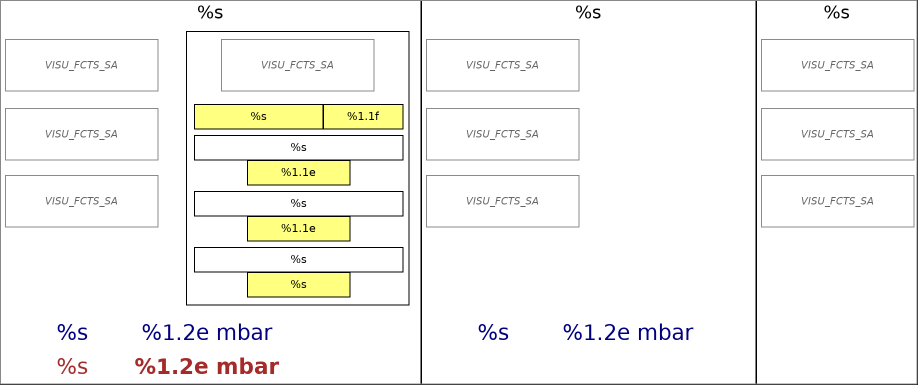
VISUALIZATION SA_POMP_2E_PCR_PPM_ASS  // 918x385
VAR_IN_OUT
	m_Input_PRG:			BLOCK_PRG_POMPAGE;
	m_Input_Jauge:			BLOCK_BCG450_ETHERCAT;
	m_Input_Process:		BLOCK_CDG_ETHERCAT;
	m_Input_Pr_Sas:			BLOCK_PCG550_ETHERCAT;
	m_Input_Vanne:			BLOCK_VVAT_650_ETHERCAT;
	m_Input_Machine:		BLOCK_MODE_MARCHE;
END_VAR
    Rectangle (0,0 421x385), "%s", text list: 'TextList_Navigation', text index: 6
    Rectangle (421,0 335x385), "%s", text list: 'TextList_Navigation', text index: 7
    Rectangle (756,0 162x385), "%s", text list: 'TextList_Navigation', text index: 13
    Frame (761,39 153x52)
        shows VISU_FCTS_SA(m_Input_ID_XML := 1, m_Input_UserRight := PRG_USER.ACTU_USER.FONCTION_SA, m_Input_Operation := m_Input_PRG.POMPAGE.OP_Marche_Pompes)
    Frame (761,108 153x52)
        shows VISU_FCTS_SA(m_Input_ID_XML := 2, m_Input_UserRight := PRG_USER.ACTU_USER.FONCTION_SA, m_Input_Operation := m_Input_PRG.POMPAGE.OP_Arret_Pompes)
    Rectangle (41,320 63x25), "%s", text variable: m_Input_Jauge.MNEMO
    Rectangle (111,318 192x29), "%1.2e mbar", text variable: m_Input_Jauge.STATE_Pression
    Rectangle (41,354 63x25), "%s", text variable: m_Input_Process.MNEMO
    Rectangle (111,352 192x29), "%1.2e mbar", text variable: m_Input_Process.STATE_Pression
    Frame (5,39 153x52)
        shows VISU_FCTS_SA(m_Input_ID_XML := 0, m_Input_UserRight := PRG_USER.ACTU_USER.FONCTION_SA, m_Input_Operation := m_Input_PRG.POMPAGE.OP_Pompage_Sec)
    Frame (426,39 153x52)
        shows VISU_FCTS_SA(m_Input_ID_XML := 0, m_Input_UserRight := PRG_USER.ACTU_USER.PRODUCTION, m_Input_Operation := m_Input_PRG.POMPAGE.OP_Pompage_SAS)
    Frame (5,108 153x52)
        shows VISU_FCTS_SA(m_Input_ID_XML := 3, m_Input_UserRight := PRG_USER.ACTU_USER.FONCTION_SA, m_Input_Operation := m_Input_PRG.POMPAGE.OP_Isolement)
    Frame (426,108 153x52)
        shows VISU_FCTS_SA(m_Input_ID_XML := 3, m_Input_UserRight := PRG_USER.ACTU_USER.FONCTION_SA, m_Input_Operation := m_Input_PRG.POMPAGE.OP_Isolement_SAS)
    Frame (761,175 153x52)
        shows VISU_FCTS_SA(m_Input_ID_XML := 17, m_Input_UserRight := PRG_USER.ACTU_USER.FONCTION_SA, m_Input_Operation := m_Input_PRG.POMPAGE.OP_Regen)
    Frame (5,175 153x52)
        shows VISU_FCTS_SA(m_Input_ID_XML := 4, m_Input_UserRight := PRG_USER.ACTU_USER.FONCTION_SA, m_Input_Operation := m_Input_PRG.POMPAGE.OP_Ventilation)
    Frame (426,175 153x52)
        shows VISU_FCTS_SA(m_Input_ID_XML := 4, m_Input_UserRight := PRG_USER.ACTU_USER.PRODUCTION, m_Input_Operation := m_Input_PRG.POMPAGE.OP_Ventilation_SAS)
    Rectangle (462,320 63x25), "%s", text variable: m_Input_Pr_Sas.MNEMO
    Rectangle (532,318 192x29), "%1.2e mbar", text variable: m_Input_Pr_Sas.STATE_Pression
    Rectangle (186,31 223x274)
    Frame (221,39 153x52)
        shows VISU_FCTS_SA(m_Input_ID_XML := 11, m_Input_UserRight := PRG_USER.ACTU_USER.FONCTION_SA, m_Input_Operation := m_Input_PRG.POMPAGE.OP_Pompage_Proc)
    RoundedRectangle (194,104 129x25), "%s", invisible if: NOT m_Input_Vanne.PRM_Mode, input disabled if: NOT (PRG_USER.ACTU_USER.FONCTION_SA AND NOT m_Input_MACHINE.STATE_Prod) OR m_Input_MACHINE.STATE_Prod, text list: 'TextList_VVAT_650_ETHERCAT', text index: 8
        OnMouseClick: toggle m_Input_Vanne.PRM_Mode
    RoundedRectangle (194,104 129x25), "%s", invisible if: m_Input_Vanne.PRM_Mode, input disabled if: NOT (PRG_USER.ACTU_USER.FONCTION_SA AND NOT m_Input_MACHINE.STATE_Prod) OR m_Input_MACHINE.STATE_Prod, text list: 'TextList_VVAT_650_ETHERCAT', text index: 7
        OnMouseClick: toggle m_Input_Vanne.PRM_Mode
    RoundedRectangle (194,135 209x25), "%s", invisible if: NOT m_Input_Vanne.PRM_Mode, text list: 'TextList_VVAT_650_ETHERCAT', text index: 4
    RoundedRectangle (194,191 209x25), "%s", invisible if: NOT m_Input_Vanne.PRM_Mode, text list: 'TextList_VVAT_650_ETHERCAT', text index: 5
    RoundedRectangle (194,247 209x25), "%s", invisible if: NOT m_Input_Vanne.PRM_Mode, text list: 'TextList_VVAT_650_ETHERCAT', text index: 6
    RoundedRectangle (247,272 103x25), "%s", text variable: m_Input_Vanne.PRM_Tim_W_Pr, invisible if: NOT m_Input_Vanne.PRM_Mode, input disabled if: NOT (PRG_USER.ACTU_USER.FONCTION_SA AND NOT m_Input_MACHINE.STATE_Prod) OR m_Input_MACHINE.STATE_Prod
        OnMouseClick: write the text variable via VisuDialogs.Keypad
    RoundedRectangle (247,216 103x25), "%1.1e", text variable: m_Input_Vanne.PRM_W_Pr_HI, invisible if: NOT m_Input_Vanne.PRM_Mode, input disabled if: NOT (PRG_USER.ACTU_USER.FONCTION_SA AND NOT m_Input_MACHINE.STATE_Prod) OR m_Input_MACHINE.STATE_Prod
        OnMouseClick: write the text variable via VisuDialogs.Numpad, min 0, max 1000
    RoundedRectangle (247,160 103x25), "%1.1e", text variable: m_Input_Vanne.PRM_W_Pr_LO, invisible if: NOT m_Input_Vanne.PRM_Mode, input disabled if: NOT (PRG_USER.ACTU_USER.FONCTION_SA AND NOT m_Input_MACHINE.STATE_Prod) OR m_Input_MACHINE.STATE_Prod
        OnMouseClick: write the text variable via VisuDialogs.Numpad, min 0, max 1000
    RoundedRectangle (323,104 80x25), "%1.1e", text variable: m_Input_Vanne.PRM_Pression, invisible if: NOT m_Input_Vanne.PRM_Mode, input disabled if: NOT (PRG_USER.ACTU_USER.FONCTION_SA AND NOT m_Input_MACHINE.STATE_Prod) OR m_Input_MACHINE.STATE_Prod
        OnMouseClick: write the text variable via VisuDialogs.Numpad, min 0, max 1000
    RoundedRectangle (323,104 80x25), "%1.1f", text variable: m_Input_Vanne.PRM_Position, invisible if: m_Input_Vanne.PRM_Mode, input disabled if: NOT (PRG_USER.ACTU_USER.FONCTION_SA AND NOT m_Input_MACHINE.STATE_Prod) OR m_Input_MACHINE.STATE_Prod
        OnMouseClick: write the text variable via VisuDialogs.Numpad, min 0, max 100
END_VISUALIZATION

(* stored: Version 1.1.0.1, ProductVersion 3.1.4024.10
   Visu SA_POMP_2E_PCR_PPM_ASS: Id {d3fa7dfe-e09f-4d1f-b521-97eeb9b3b50c} *)
